PROGRAM BarCodeReaders
VAR
	BCR_S6040_01: CognexDataMan260;		// P8005 Induct Confirm
	BCR_S7004_01: CognexDataMan260;		// P8010 Location Update
			
		
	Arrival_Item 			: ST_Item;		// Output Item (Bar code read) To Sort PLC
	LastArrival_Item		: ST_Item;		// Last Output Item (Bar code read) To Sort PLC
	ReadID_P6040_Old		: UDINT;

	st_SorterArrivalBuffer AT %Q*	: ST_ItemBuffer;		// Output from the Barcode Reader to the sorter
	st_ArrivalFdbkIn AT %I*			: ST_ItemBufferFdbk;
	st_ArrivalFdbkOut 				: ST_ItemBufferFdbk;
	fb_SorterArrivalBuffer			: FB_ItemBuffer;	// Function to Process the SorterArrivalBuffer
	
	sBcr_S6040_01Log			: STRING;
	tpBcr_S6040_01Trig					: TP;	// Pulse timer for BCR Reader

	rSorterPE					: R_TRIG; 	// Capture the Rising edge of the Sorter BCR PE
	fSorterPE					: F_TRIG; 	// Capture the Falling edge of the Sorter BCR PE
	r_BCR_S6040_01TriggerON			: R_TRIG;
	f_BCR_S6040_01TriggerON			: F_TRIG;

END_VAR

// Create instances of Buffer Processing Functions to initialize the buffers and data
fb_SorterArrivalBuffer.Master := TRUE;

// Setup Logging
fb_SorterArrivalBuffer.LogEntries := .nItemBufferLogEnable.ARRIVALS;

// Setup Buffer Name for Logging
fb_SorterArrivalBuffer.Name := 'SYS ARRIVAL';

fb_SorterArrivalBuffer(st_BufferData := st_SorterArrivalBuffer
					, st_BufferFdbkIn := st_ArrivalFdbkIn
					, st_BufferFdbkOut => st_ArrivalFdbkOut);

IF GVL_IO.INIT THEN
	fb_SorterArrivalBuffer.Clear();
END_IF
// Reset All Metrics when requested
IF MAIN.In_ResetAllMetrics THEN
	BCR_S6040_01.In_ResetCounts := MAIN.In_ResetAllMetrics;
	BCR_S7004_01.In_ResetCounts := MAIN.In_ResetAllMetrics;
END_IF

// Set up Bar Code Readers
//----------------------------------------P6040--------------------------------------------------------------
BCR_S6040_01.LogEntries := .nBarcodeLogEnable.BCR_S6040_01_LOG;
BCR_S6040_01(
	In_ReadTrig:= PhotoEyes.PE_6261.Out_OnFltrd, 
	In_ResetCounts:= , 
	In_TriggerOnTime := T#20MS ,
	In_EquipID := '00001',
	Out_NewReadTrig=> , 
	Out_ReadString=> , 
	Out_ReadStatus=> ,
	Out_ResultID=>, 
	MisreadCount=> , 
	GoodreadCount=> );
	
BCR_S6040_01.LogEntries := .nBarcodeLogEnable.BCR_S6040_01_LOG;
tpBcr_S6040_01Trig(
	IN := PhotoEyes.PE_6261.Out,
				PT := T#10MS,
				Q =>);
// Capture rising and falling edge Triggers of the Sorter BCR Trigger PE
 rSorterPE(CLK:= PhotoEyes.PE_6261.Out, Q =>);
 fSorterPE(CLK:= PhotoEyes.PE_6261.Out, Q =>);

// Log the rising edge of the Trigger
IF rSorterPE.Q THEN
	IF nBarcodeLogEnable.TRIGGER_PE THEN
		// Write to the Error List
		ADSLOGSTR( msgCtrlMask := ADSLOG_MSGTYPE_HINT OR ADSLOG_MSGTYPE_LOG,
			msgFmtStr := 'Sort BCR PE Blocked : %s',
			strArg := BOOL_TO_STRING(PhotoEyes.PE_6261.Out)
			); 
	END_IF
END_IF

// Log the falling edge of the Trigger
IF fSorterPE.Q THEN
	IF nBarcodeLogEnable.TRIGGER_PE THEN
		// Write to the Error List
		ADSLOGSTR( msgCtrlMask := ADSLOG_MSGTYPE_HINT OR ADSLOG_MSGTYPE_LOG,
			msgFmtStr := 'Sort BCR PE Blocked : %s',
			strArg := BOOL_TO_STRING(PhotoEyes.PE_6261.Out)
		);
	END_IF
END_IF


// Capture rising and falling edge Triggers of the Sorter BCR Trigger PE
r_BCR_S6040_01TriggerOn(CLK:= BCR_S6040_01.Out_TriggerState, Q =>);
f_BCR_S6040_01TriggerOn(CLK:= BCR_S6040_01.Out_TriggerState, Q =>);

// Log the rising edge of the Trigger
IF r_BCR_S6040_01TriggerOn.Q THEN
	IF nBarcodeLogEnable.TRIGGER THEN
		// Write to the Error List
		ADSLOGSTR( msgCtrlMask := ADSLOG_MSGTYPE_HINT OR ADSLOG_MSGTYPE_LOG
			, msgFmtStr := 'Sort BCR Trigger : %s'
			, strArg := BOOL_TO_STRING(BCR_S6040_01.Out_TriggerState)); 
	END_IF
END_IF


// Send Read Information to Sorter	
//	Creates Arrival message at sorter
IF ReadID_P6040_Old <> BarCodeReaders.BCR_S6040_01.GoodreadCount THEN
	Arrival_Item.UniqueID := BCR_S6040_01.Out_ResultID;
	Arrival_Item.ID := BCR_S6040_01.Out_ReadString;
	Arrival_Item.Status := E_StatusCode.UpdateRequested;
	Arrival_Item.DeviceID := GVL_IO.SorterName;
	Arrival_Item.MessageType := E_MessageIds.Arrival_23;
	Arrival_Item.Destination := MsgControl.DefDestination;
	Arrival_Item.Length := 0;
	LastArrival_Item := Arrival_Item;
	fb_SorterArrivalBuffer.AddItem(Arrival_Item);
	ReadID_P6040_Old := BarCodeReaders.BCR_S6040_01.GoodreadCount;
ELSE 
	Arrival_Item := MsgControl.BlankItem;
	Arrival_Item.Status := E_StatusCode.UpdateRequested;
END_IF	

//----------------------------------------P7004--------------------------------------------------------------	
BCR_S7004_01.LogEntries := .nBarcodeLogEnable.BCR_S7004_01_LOG;
BCR_S7004_01(
	In_ReadTrig:= PhotoEyes.PE_12221.Out_OnFltrd, 
	In_ResetCounts:= , 
	In_TriggerOnTime := T#20MS ,
	In_EquipID := '00002',
	Out_NewReadTrig=> , 
	Out_ReadString=> , 
	Out_ReadStatus=> ,
	Out_ResultID=>, 
	MisreadCount=> , 
	GoodreadCount=> );

END_PROGRAM

(* stored: Version 1.1.0.1, ProductVersion 3.1.4024.4
   POU BarCodeReaders: Id {6db726c2-b8f2-4f56-a606-779b1afe45e4}, SpecialFunc None *)
